// LS Electric XG5000 project: day13
// PLC LSPLC
// module base 0 slot 0: 입출력 모듈:XBC-DR30S (DC 24V 입력 18점, 릴레이 출력 12점)

PROGRAM day13 (task: 스캔 프로그램)

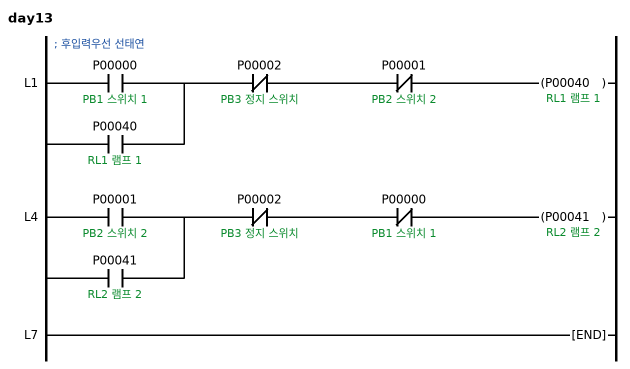
// 후입력우선 선태연
; L1
LOAD      P00000	// PB1 스위치 1
OR        P00040	// RL1 램프 1
AND NOT   P00002	// PB3 정지 스위치
AND NOT   P00001	// PB2 스위치 2
OUT       P00040	// RL1 램프 1
; L4
LOAD      P00001	// PB2 스위치 2
OR        P00041	// RL2 램프 2
AND NOT   P00002	// PB3 정지 스위치
AND NOT   P00000	// PB1 스위치 1
OUT       P00041	// RL2 램프 2
; L7
END